(* Logix 5000 project; controller GEA_Test_Chamber vendor 1 type 14 code 196 rev 32.14; software revision 32.04; part 6 of 11 *)
(* tags used below, declared in another part *)
   bPulse05Hz : BOOL;
   bPulse0_1Hz : BOOL;
   bPulse10Hz : BOOL;
   bPulse1Hz : BOOL;
   Cycle_Counter : SINT;
   FVIR_1_S_Step : INT;
   FVIR_1_W_Step : INT;
   FVIR_2_S_Step : INT;
   FVIR_2_W_Step : INT;
   FVIR_3_S_Step : INT;
   FVIR_3_W_Step : INT;
   FVIR_4_S_Step : INT;
   FVIR_4_W_Step : INT;
   FVIR_Gas_Flow_Heater_Indication_1 : BOOL;
   FVIR_Gas_Flow_Heater_Indication_2 : BOOL;
   FVIR_Gas_SCPM_FI001 : REAL;
   FVIR_Gas_SCPM_FI0012 : REAL;
   FVIR_LabView_Comm_OK : BOOL;
   FVIR_Water_Outler_Flow : REAL;
   Gasoline_Step : SINT;
   Mannequin_GoTo_Home : BOOL;
   Mannequin_GoTo_Work : BOOL;
   Mannequin_Step : DINT;
   Pulse : BOOL[32];
   Spill_GoTo_Home : BOOL;
   Spill_GoTo_Work : BOOL;
   Start_Manequinn_Move : BOOL;
   Start_Manequinn_Seq : BOOL;
   Start_Manequinn_Seq_Man : BOOL;
   Start_Spill_Gasoline : BOOL;
   Tigger_First_Manniquine_Seq : BOOL;
   Timer_Delay : TIMER[30];
   tof0_1sPulse : TIMER;
   tof10sPulse : TIMER;
   tof1sPulse : TIMER;
   tof2sPulse : TIMER;
   ton0_1sPulse : TIMER;
   ton10sPulse : TIMER;
   ton1sPulse : TIMER;
   ton2sPulse : TIMER;
   TON_LifeBit_OFF : TIMER;
   TON_LifeBit_ON : TIMER;
   Water_Outlet_Flow_OK : BOOL;
   Water_Outlet_Valve : INT;
   Control_Off : BOOL;
   FVIR_Error_MSG : INT;
   FVIR_LabView_Control : INT;
   FVIR_LabView_Status : INT;
   FVIR_Mannequin_Direction_TimeDelay : INT;
   FVIR_Mannequin_Time_Pause : INT;
   FVIR_Number_Mannequin_Movement : INT;
   FVIR_Reset_Cnt_inprogress : BOOL;
   Output_FVIR : Output_FVIR;
   SET_0 : BOOL;
   SET_1 : BOOL;
(* FVIR_Chamber, continued *)

ROUTINE FVIR_Main   (* ladder *)
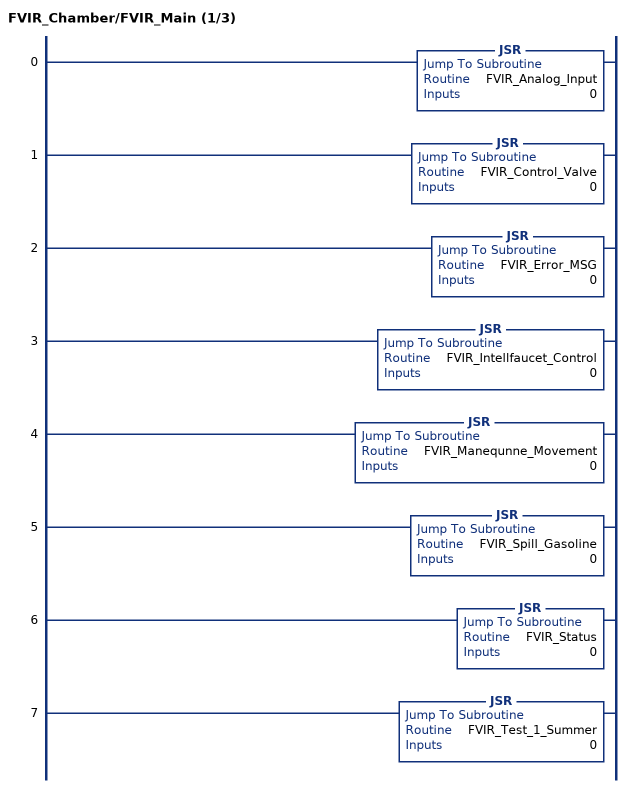
   0: JSR(FVIR_Analog_Input,0);
   1: JSR(FVIR_Control_Valve,0);
   2: JSR(FVIR_Error_MSG,0);
   3: JSR(FVIR_Intellfaucet_Control,0);
   4: JSR(FVIR_Manequnne_Movement,0);
   5: JSR(FVIR_Spill_Gasoline,0);
   6: JSR(FVIR_Status,0);
   7: JSR(FVIR_Test_1_Summer,0);
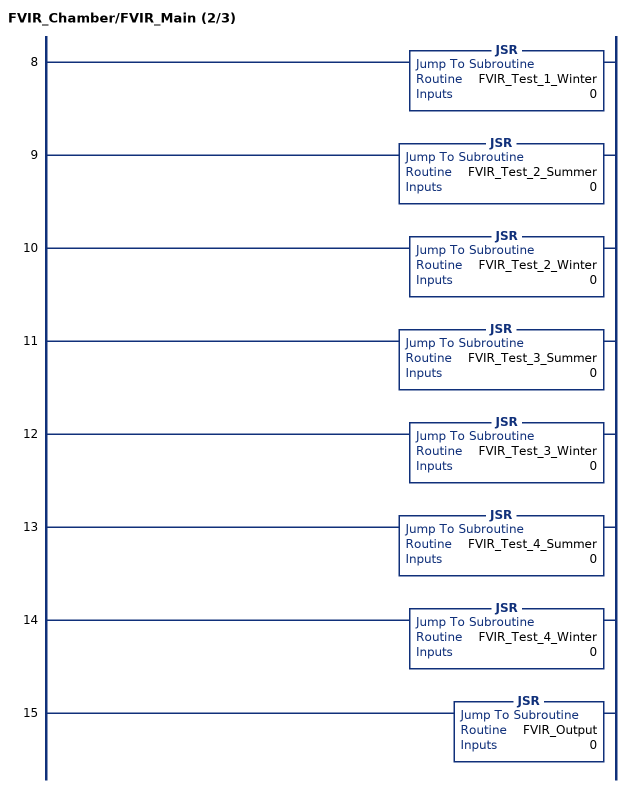
   8: JSR(FVIR_Test_1_Winter,0);
   9: JSR(FVIR_Test_2_Summer,0);
   10: JSR(FVIR_Test_2_Winter,0);
   11: JSR(FVIR_Test_3_Summer,0);
   12: JSR(FVIR_Test_3_Winter,0);
   13: JSR(FVIR_Test_4_Summer,0);
   14: JSR(FVIR_Test_4_Winter,0);
   15: JSR(FVIR_Output,0);
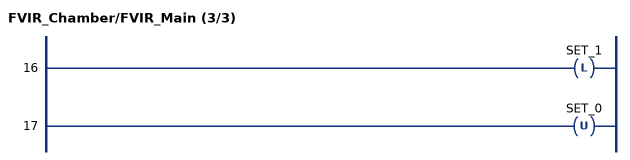
   16: OTL(SET_1);
   17: OTU(SET_0);
END_ROUTINE

ROUTINE FVIR_Manequnne_Movement   (* ladder *)
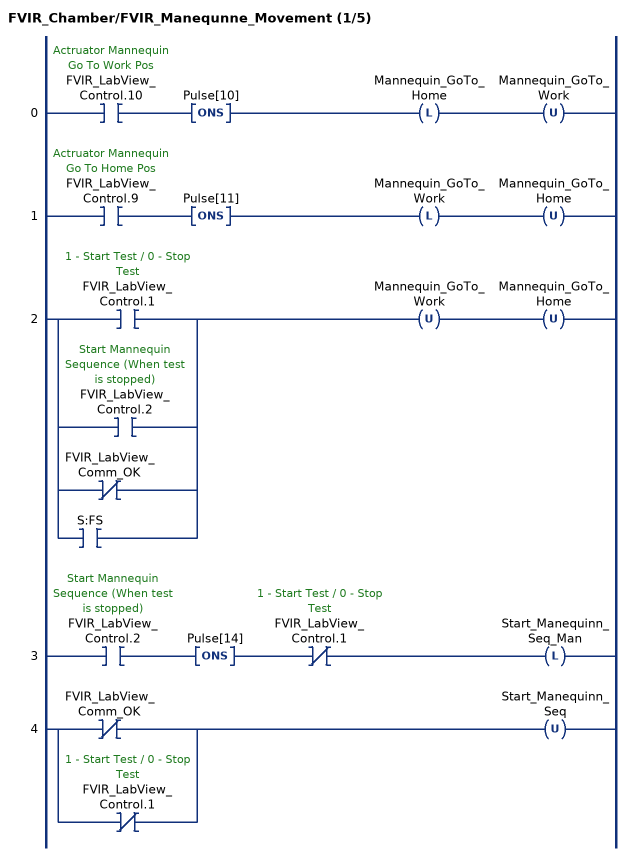
   0: XIC(FVIR_LabView_Control.10)ONS(Pulse[10])OTL(Mannequin_GoTo_Home)OTU(Mannequin_GoTo_Work);
   1: XIC(FVIR_LabView_Control.9)ONS(Pulse[11])OTL(Mannequin_GoTo_Work)OTU(Mannequin_GoTo_Home);
   2: [XIC(FVIR_LabView_Control.1) ,XIC(FVIR_LabView_Control.2) ,[XIO(FVIR_LabView_Comm_OK) ,XIC(S:FS) ] ]OTU(Mannequin_GoTo_Work)OTU(Mannequin_GoTo_Home);
   3: XIC(FVIR_LabView_Control.2)ONS(Pulse[14])XIO(FVIR_LabView_Control.1)OTL(Start_Manequinn_Seq_Man);
   4: [XIO(FVIR_LabView_Comm_OK) ,XIO(FVIR_LabView_Control.1) ]OTU(Start_Manequinn_Seq);
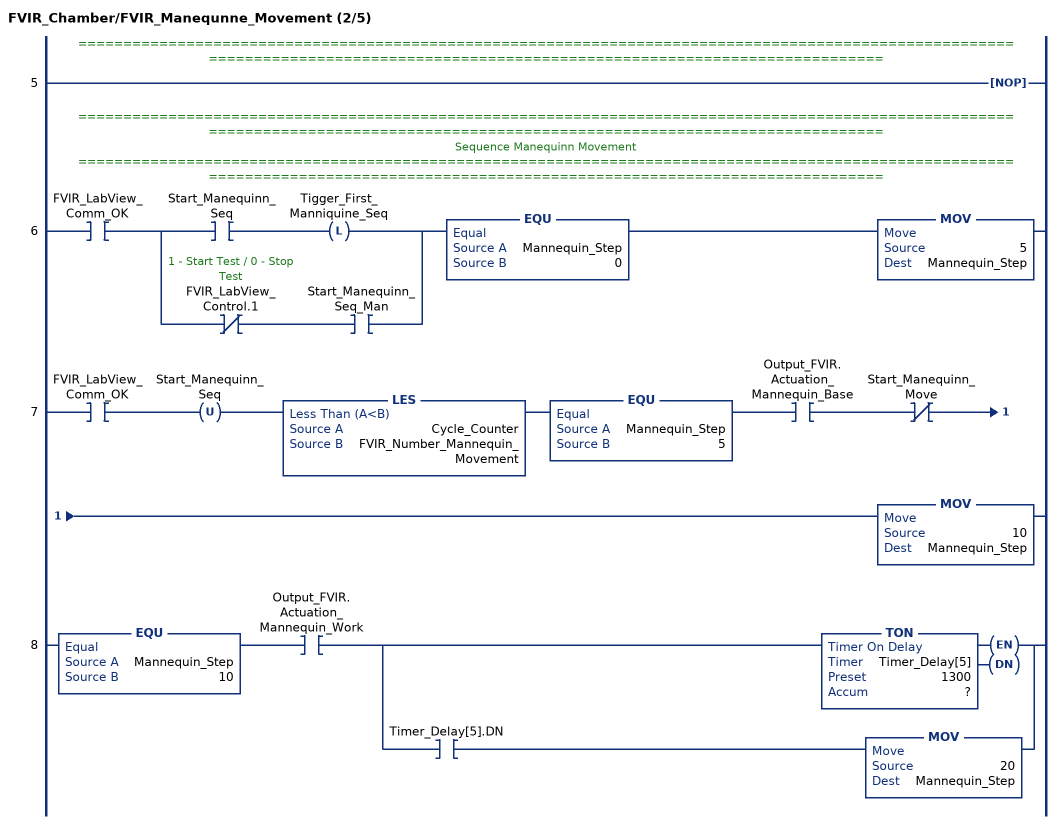
   // ===================================================================================================================================================================================
   5: NOP();
   // ===================================================================================================================================================================================
   // Sequence Manequinn Movement
   // ===================================================================================================================================================================================
   6: XIC(FVIR_LabView_Comm_OK)[XIC(Start_Manequinn_Seq) OTL(Tigger_First_Manniquine_Seq) ,XIO(FVIR_LabView_Control.1) XIC(Start_Manequinn_Seq_Man) ]EQU(Mannequin_Step,0)MOV(5,Mannequin_Step);
   7: XIC(FVIR_LabView_Comm_OK)OTU(Start_Manequinn_Seq)LES(Cycle_Counter,FVIR_Number_Mannequin_Movement)EQU(Mannequin_Step,5)XIC(Output_FVIR.Actuation_Mannequin_Base)XIO(Start_Manequinn_Move)MOV(10,Mannequin_Step);
   8: EQU(Mannequin_Step,10)XIC(Output_FVIR.Actuation_Mannequin_Work)[TON(Timer_Delay[5],?,?) ,XIC(Timer_Delay[5].DN) MOV(20,Mannequin_Step) ];
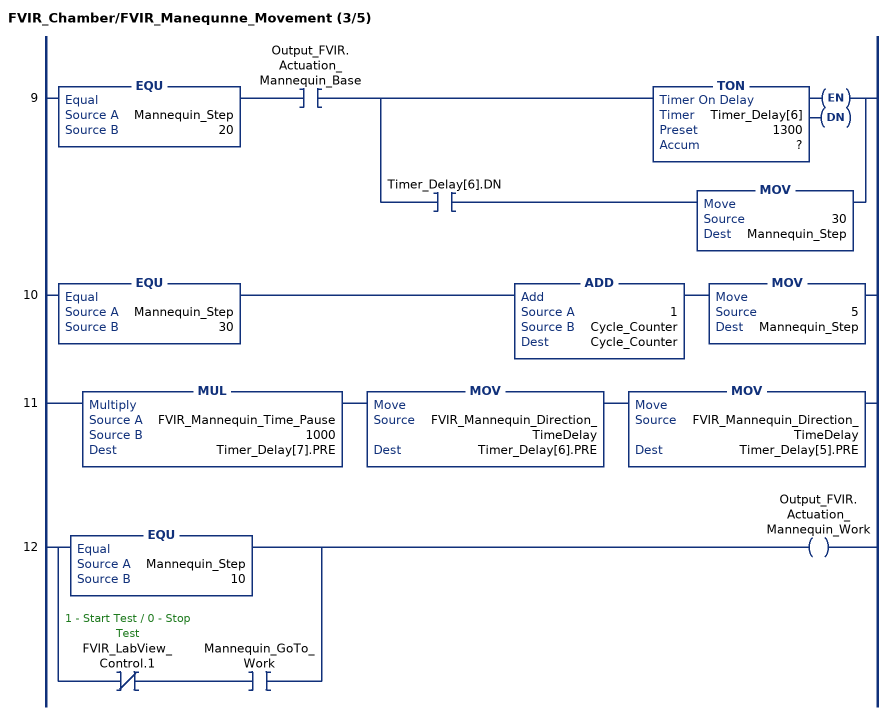
   9: EQU(Mannequin_Step,20)XIC(Output_FVIR.Actuation_Mannequin_Base)[TON(Timer_Delay[6],?,?) ,XIC(Timer_Delay[6].DN) MOV(30,Mannequin_Step) ];
   10: EQU(Mannequin_Step,30)ADD(1,Cycle_Counter,Cycle_Counter)MOV(5,Mannequin_Step);
   11: MUL(FVIR_Mannequin_Time_Pause,1000,Timer_Delay[7].PRE)MOV(FVIR_Mannequin_Direction_TimeDelay,Timer_Delay[6].PRE)MOV(FVIR_Mannequin_Direction_TimeDelay,Timer_Delay[5].PRE);
   12: [EQU(Mannequin_Step,10) ,XIO(FVIR_LabView_Control.1) XIC(Mannequin_GoTo_Work) ]OTE(Output_FVIR.Actuation_Mannequin_Work);
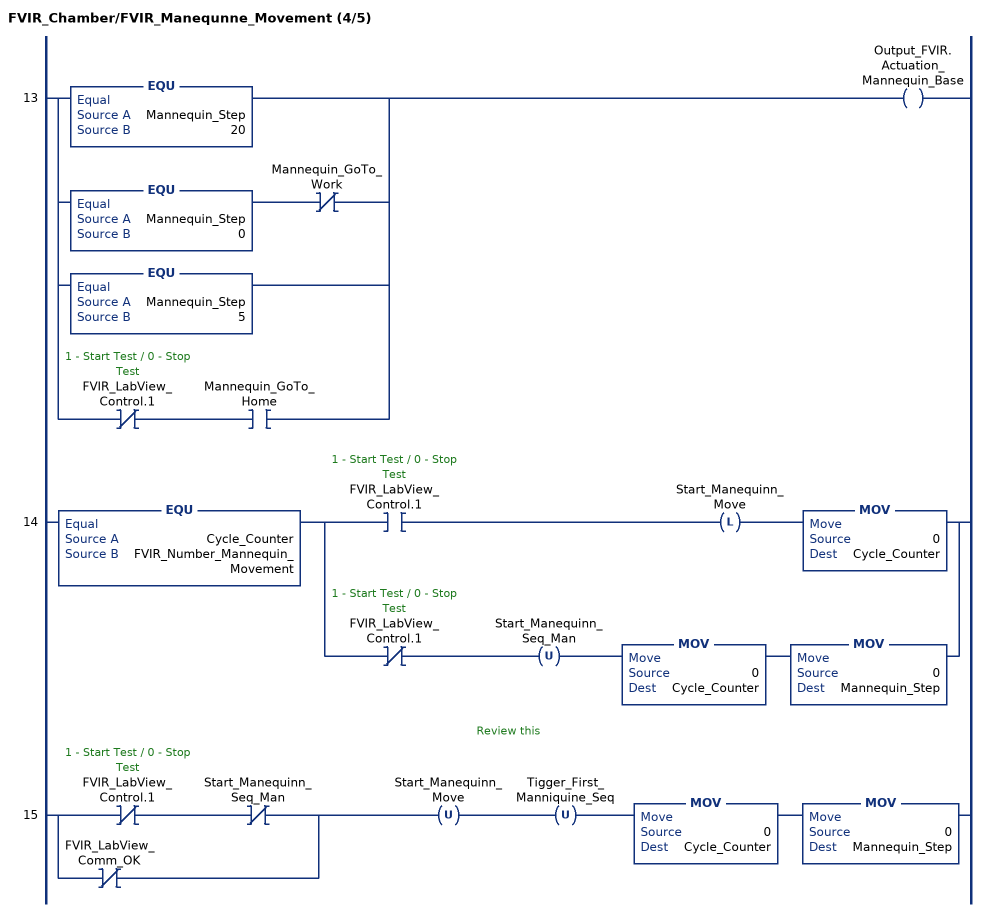
   13: [EQU(Mannequin_Step,20) ,[[EQU(Mannequin_Step,0) XIO(Mannequin_GoTo_Work) ,EQU(Mannequin_Step,5) ] ,XIO(FVIR_LabView_Control.1) XIC(Mannequin_GoTo_Home) ] ]OTE(Output_FVIR.Actuation_Mannequin_Base);
   14: EQU(Cycle_Counter,FVIR_Number_Mannequin_Movement)[XIC(FVIR_LabView_Control.1) OTL(Start_Manequinn_Move) MOV(0,Cycle_Counter) ,XIO(FVIR_LabView_Control.1) OTU(Start_Manequinn_Seq_Man) MOV(0,Cycle_Counter) MOV(0,Mannequin_Step) ];
   // Review this
   15: [XIO(FVIR_LabView_Control.1) XIO(Start_Manequinn_Seq_Man) ,XIO(FVIR_LabView_Comm_OK) ]OTU(Start_Manequinn_Move)OTU(Tigger_First_Manniquine_Seq)MOV(0,Cycle_Counter)MOV(0,Mannequin_Step);
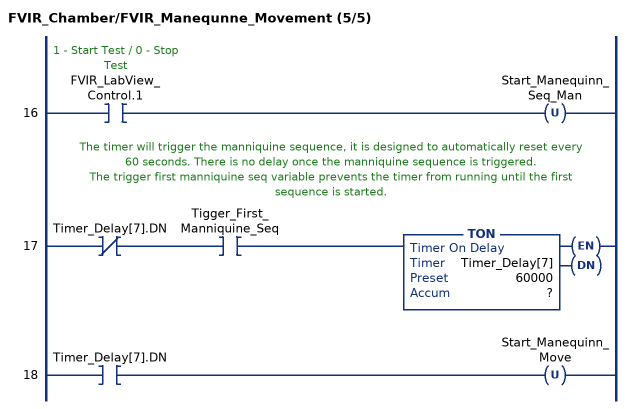
   16: XIC(FVIR_LabView_Control.1)OTU(Start_Manequinn_Seq_Man);
   // The timer will trigger the manniquine sequence, it is designed to automatically reset every 60 seconds. There is no delay once the manniquine sequence is triggered.
   //  The trigger first manniquine seq variable prevents the timer from running until the first sequence is started.
   17: XIO(Timer_Delay[7].DN)XIC(Tigger_First_Manniquine_Seq)TON(Timer_Delay[7],?,?);
   18: XIC(Timer_Delay[7].DN)OTU(Start_Manequinn_Move);
END_ROUTINE

ROUTINE FVIR_Output   (* ladder *)
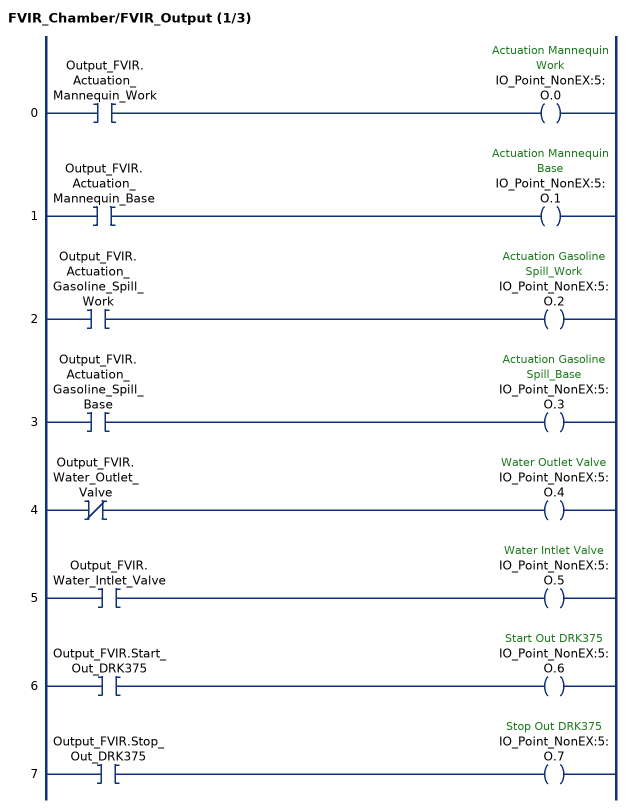
   0: XIC(Output_FVIR.Actuation_Mannequin_Work)OTE(IO_Point_NonEX:5:O.0);
   1: XIC(Output_FVIR.Actuation_Mannequin_Base)OTE(IO_Point_NonEX:5:O.1);
   2: XIC(Output_FVIR.Actuation_Gasoline_Spill_Work)OTE(IO_Point_NonEX:5:O.2);
   3: XIC(Output_FVIR.Actuation_Gasoline_Spill_Base)OTE(IO_Point_NonEX:5:O.3);
   4: XIO(Output_FVIR.Water_Outlet_Valve)OTE(IO_Point_NonEX:5:O.4);
   5: XIC(Output_FVIR.Water_Intlet_Valve)OTE(IO_Point_NonEX:5:O.5);
   6: XIC(Output_FVIR.Start_Out_DRK375)OTE(IO_Point_NonEX:5:O.6);
   7: XIC(Output_FVIR.Stop_Out_DRK375)OTE(IO_Point_NonEX:5:O.7);
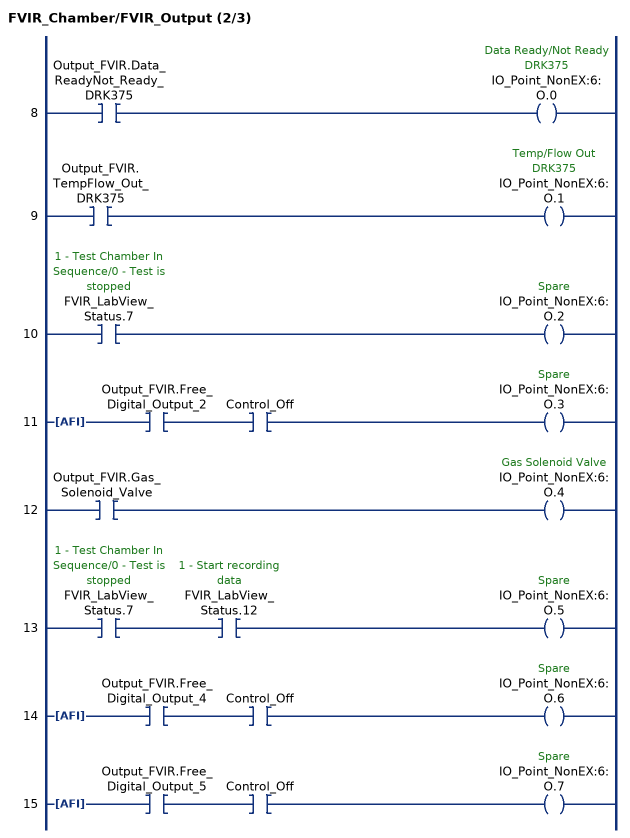
   8: XIC(Output_FVIR.Data_ReadyNot_Ready_DRK375)OTE(IO_Point_NonEX:6:O.0);
   9: XIC(Output_FVIR.TempFlow_Out_DRK375)OTE(IO_Point_NonEX:6:O.1);
   10: XIC(FVIR_LabView_Status.7)OTE(IO_Point_NonEX:6:O.2);
   11: AFI()XIC(Output_FVIR.Free_Digital_Output_2)XIC(Control_Off)OTE(IO_Point_NonEX:6:O.3);
   12: XIC(Output_FVIR.Gas_Solenoid_Valve)OTE(IO_Point_NonEX:6:O.4);
   13: XIC(FVIR_LabView_Status.7)XIC(FVIR_LabView_Status.12)OTE(IO_Point_NonEX:6:O.5);
   14: AFI()XIC(Output_FVIR.Free_Digital_Output_4)XIC(Control_Off)OTE(IO_Point_NonEX:6:O.6);
   15: AFI()XIC(Output_FVIR.Free_Digital_Output_5)XIC(Control_Off)OTE(IO_Point_NonEX:6:O.7);
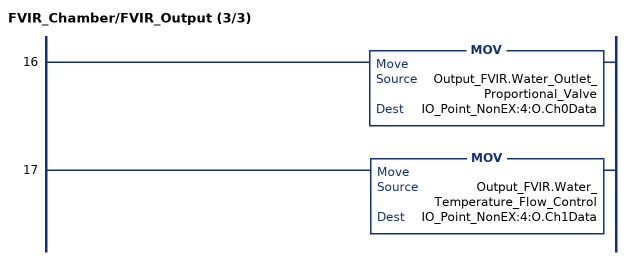
   16: MOV(Output_FVIR.Water_Outlet_Proportional_Valve,IO_Point_NonEX:4:O.Ch0Data);
   17: MOV(Output_FVIR.Water_Temperature_Flow_Control,IO_Point_NonEX:4:O.Ch1Data);
END_ROUTINE

ROUTINE FVIR_Spill_Gasoline   (* ladder *)
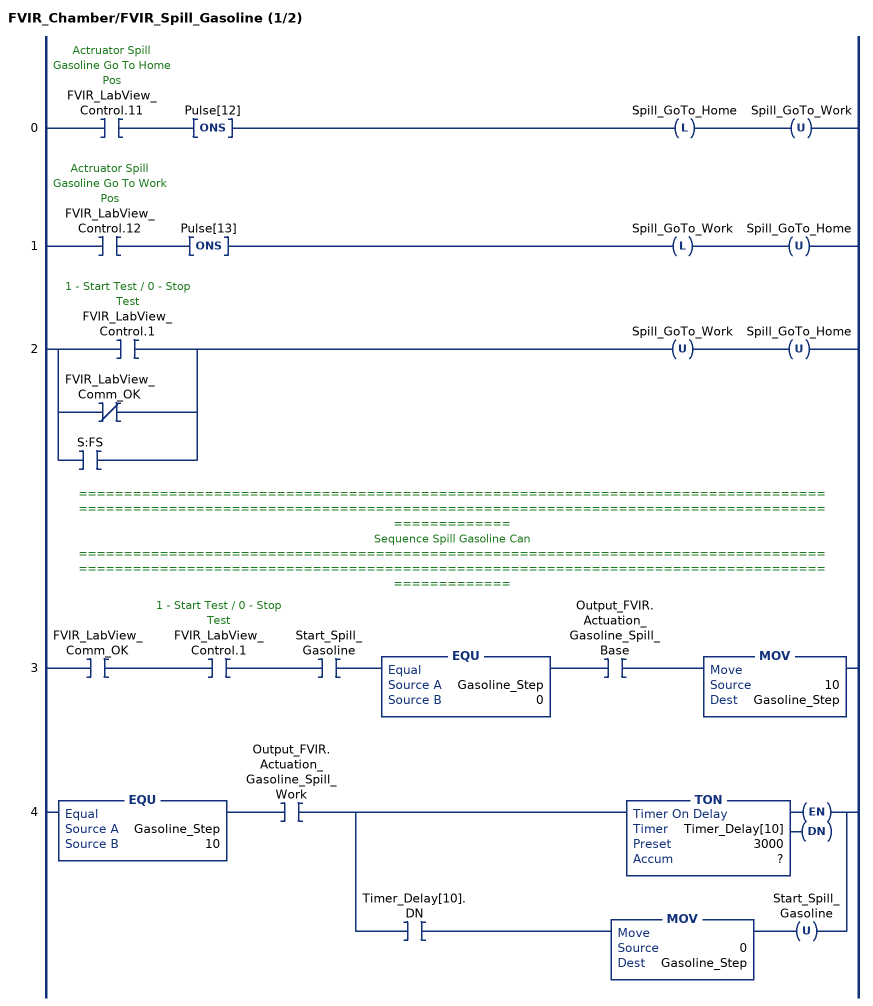
   0: XIC(FVIR_LabView_Control.11)ONS(Pulse[12])OTL(Spill_GoTo_Home)OTU(Spill_GoTo_Work);
   1: XIC(FVIR_LabView_Control.12)ONS(Pulse[13])OTL(Spill_GoTo_Work)OTU(Spill_GoTo_Home);
   2: [XIC(FVIR_LabView_Control.1) ,[XIO(FVIR_LabView_Comm_OK) ,XIC(S:FS) ] ]OTU(Spill_GoTo_Work)OTU(Spill_GoTo_Home);
   // ===================================================================================================================================================================================
   // Sequence Spill Gasoline Can
   // ===================================================================================================================================================================================
   3: XIC(FVIR_LabView_Comm_OK)XIC(FVIR_LabView_Control.1)XIC(Start_Spill_Gasoline)EQU(Gasoline_Step,0)XIC(Output_FVIR.Actuation_Gasoline_Spill_Base)MOV(10,Gasoline_Step);
   4: EQU(Gasoline_Step,10)XIC(Output_FVIR.Actuation_Gasoline_Spill_Work)[TON(Timer_Delay[10],?,?) ,XIC(Timer_Delay[10].DN) MOV(0,Gasoline_Step) OTU(Start_Spill_Gasoline) ];
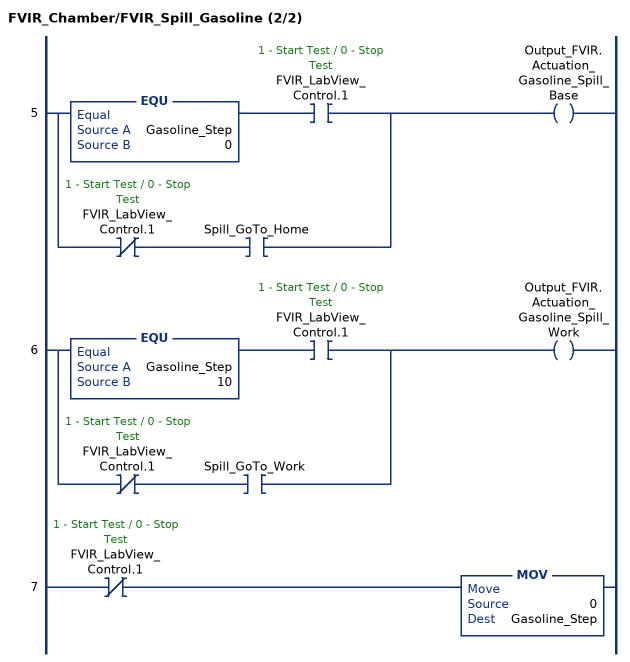
   5: [EQU(Gasoline_Step,0) XIC(FVIR_LabView_Control.1) ,XIO(FVIR_LabView_Control.1) XIC(Spill_GoTo_Home) ]OTE(Output_FVIR.Actuation_Gasoline_Spill_Base);
   6: [EQU(Gasoline_Step,10) XIC(FVIR_LabView_Control.1) ,XIO(FVIR_LabView_Control.1) XIC(Spill_GoTo_Work) ]OTE(Output_FVIR.Actuation_Gasoline_Spill_Work);
   7: XIO(FVIR_LabView_Control.1)MOV(0,Gasoline_Step);
END_ROUTINE

ROUTINE FVIR_Status   (* ladder *)
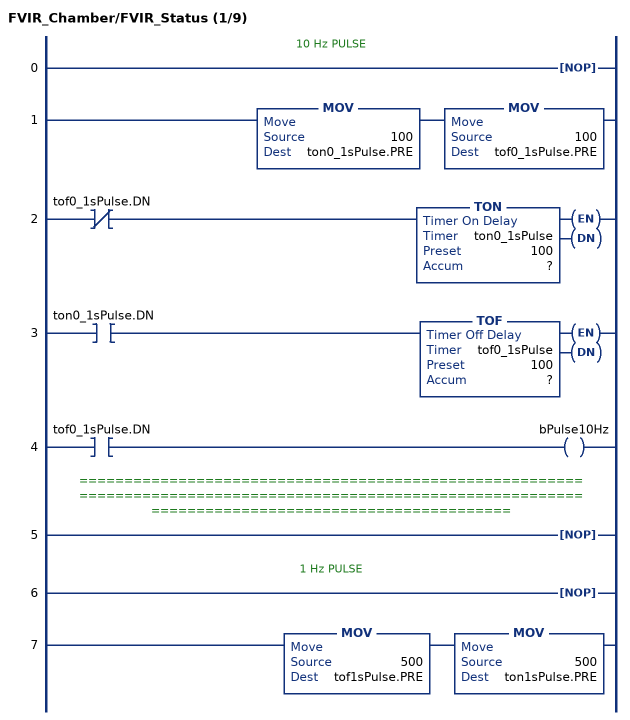
   // 10 Hz PULSE
   0: NOP();
   1: MOV(100,ton0_1sPulse.PRE)MOV(100,tof0_1sPulse.PRE);
   2: XIO(tof0_1sPulse.DN)TON(ton0_1sPulse,?,?);
   3: XIC(ton0_1sPulse.DN)TOF(tof0_1sPulse,?,?);
   4: XIC(tof0_1sPulse.DN)OTE(bPulse10Hz);
   // ========================================================================================================================================================
   5: NOP();
   // 1 Hz PULSE
   6: NOP();
   7: MOV(500,tof1sPulse.PRE)MOV(500,ton1sPulse.PRE);
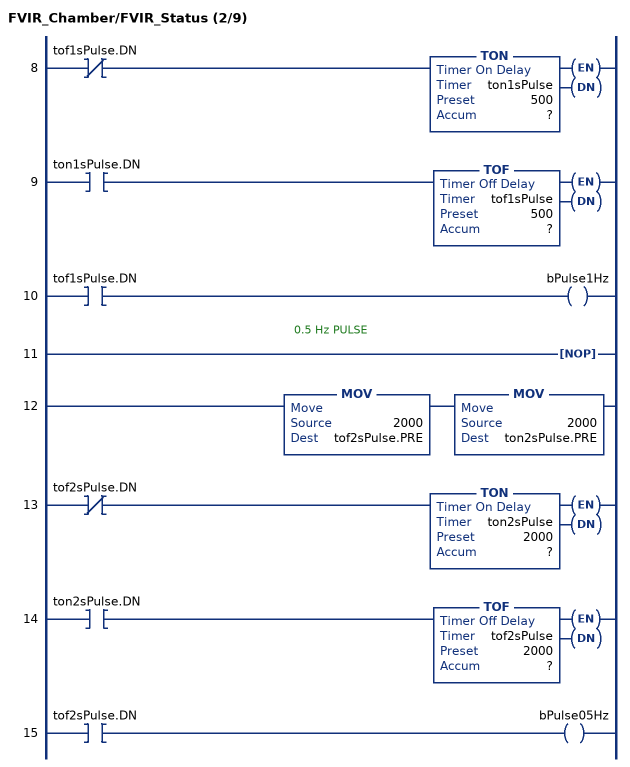
   8: XIO(tof1sPulse.DN)TON(ton1sPulse,?,?);
   9: XIC(ton1sPulse.DN)TOF(tof1sPulse,?,?);
   10: XIC(tof1sPulse.DN)OTE(bPulse1Hz);
   // 0.5 Hz PULSE
   11: NOP();
   12: MOV(2000,tof2sPulse.PRE)MOV(2000,ton2sPulse.PRE);
   13: XIO(tof2sPulse.DN)TON(ton2sPulse,?,?);
   14: XIC(ton2sPulse.DN)TOF(tof2sPulse,?,?);
   15: XIC(tof2sPulse.DN)OTE(bPulse05Hz);
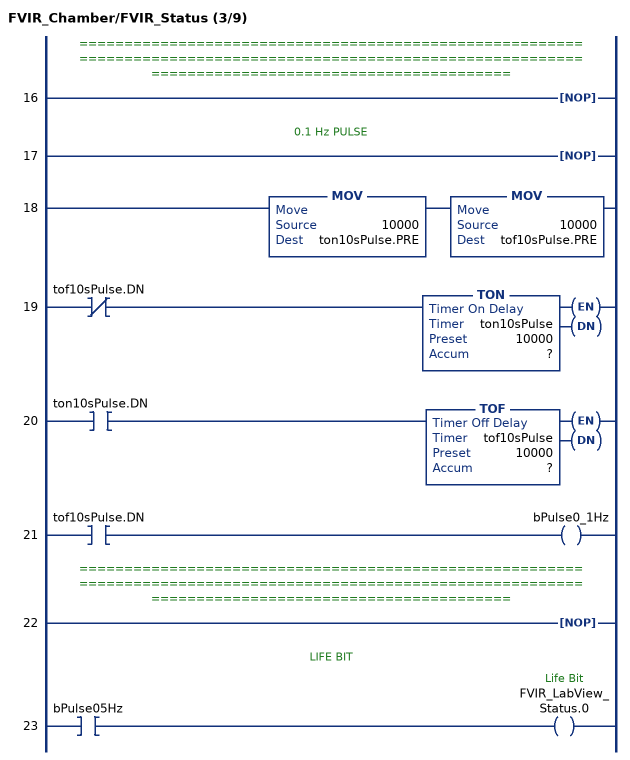
   // ========================================================================================================================================================
   16: NOP();
   // 0.1 Hz PULSE
   17: NOP();
   18: MOV(10000,ton10sPulse.PRE)MOV(10000,tof10sPulse.PRE);
   19: XIO(tof10sPulse.DN)TON(ton10sPulse,?,?);
   20: XIC(ton10sPulse.DN)TOF(tof10sPulse,?,?);
   21: XIC(tof10sPulse.DN)OTE(bPulse0_1Hz);
   // ========================================================================================================================================================
   22: NOP();
   // LIFE BIT
   23: XIC(bPulse05Hz)OTE(FVIR_LabView_Status.0);
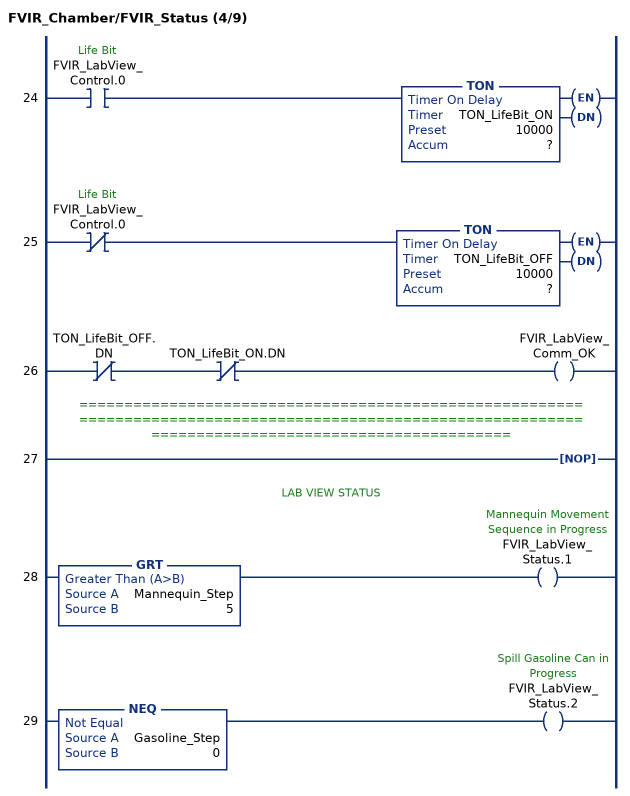
   24: XIC(FVIR_LabView_Control.0)TON(TON_LifeBit_ON,?,?);
   25: XIO(FVIR_LabView_Control.0)TON(TON_LifeBit_OFF,?,?);
   26: XIO(TON_LifeBit_OFF.DN)XIO(TON_LifeBit_ON.DN)OTE(FVIR_LabView_Comm_OK);
   // ========================================================================================================================================================
   27: NOP();
   // LAB VIEW STATUS
   28: GRT(Mannequin_Step,5)OTE(FVIR_LabView_Status.1);
   29: NEQ(Gasoline_Step,0)OTE(FVIR_LabView_Status.2);
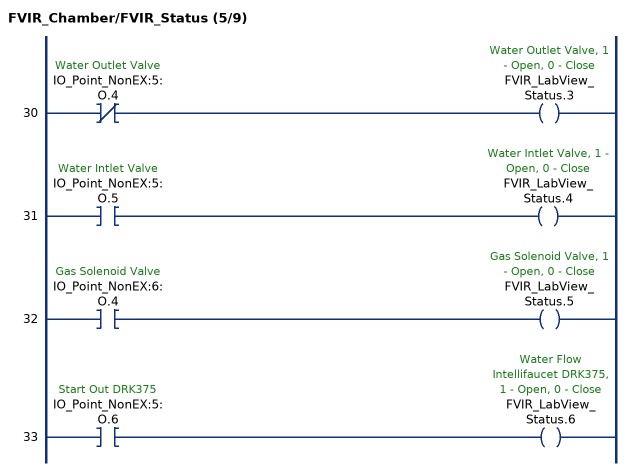
   30: XIO(IO_Point_NonEX:5:O.4)OTE(FVIR_LabView_Status.3);
   31: XIC(IO_Point_NonEX:5:O.5)OTE(FVIR_LabView_Status.4);
   32: XIC(IO_Point_NonEX:6:O.4)OTE(FVIR_LabView_Status.5);
   33: XIC(IO_Point_NonEX:5:O.6)OTE(FVIR_LabView_Status.6);
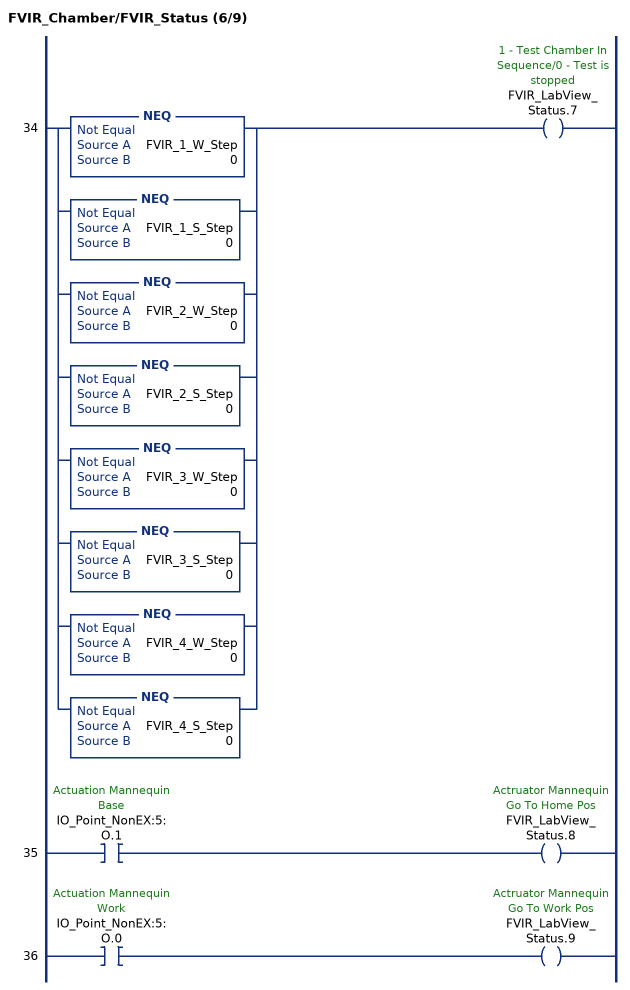
   34: [NEQ(FVIR_1_W_Step,0) ,NEQ(FVIR_1_S_Step,0) ,NEQ(FVIR_2_W_Step,0) ,NEQ(FVIR_2_S_Step,0) ,NEQ(FVIR_3_W_Step,0) ,NEQ(FVIR_3_S_Step,0) ,NEQ(FVIR_4_W_Step,0) ,NEQ(FVIR_4_S_Step,0) ]OTE(FVIR_LabView_Status.7);
   35: XIC(IO_Point_NonEX:5:O.1)OTE(FVIR_LabView_Status.8);
   36: XIC(IO_Point_NonEX:5:O.0)OTE(FVIR_LabView_Status.9);
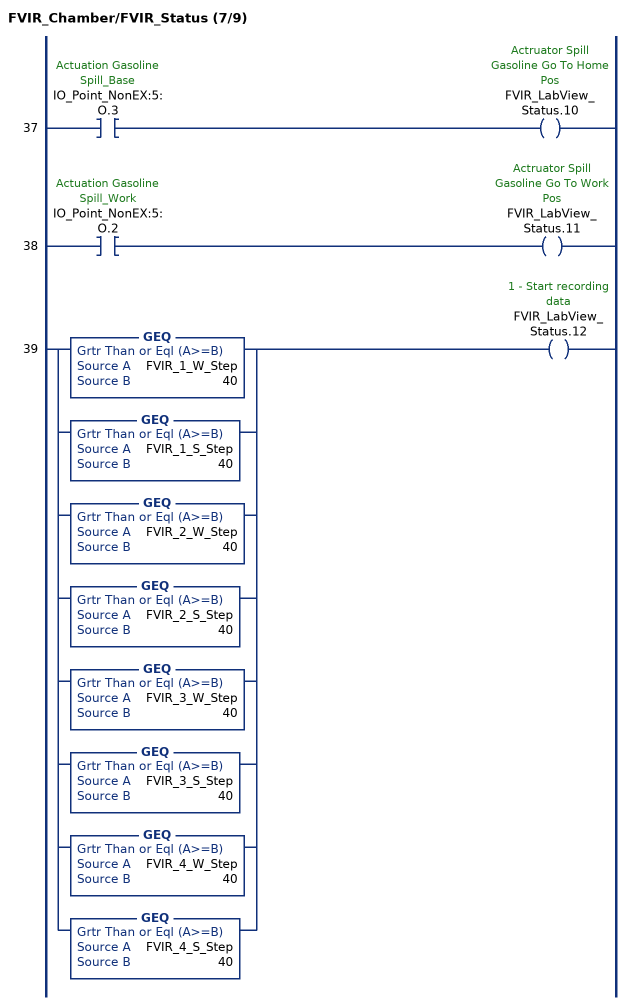
   37: XIC(IO_Point_NonEX:5:O.3)OTE(FVIR_LabView_Status.10);
   38: XIC(IO_Point_NonEX:5:O.2)OTE(FVIR_LabView_Status.11);
   39: [GEQ(FVIR_1_W_Step,40) ,GEQ(FVIR_1_S_Step,40) ,GEQ(FVIR_2_W_Step,40) ,GEQ(FVIR_2_S_Step,40) ,GEQ(FVIR_3_W_Step,40) ,GEQ(FVIR_3_S_Step,40) ,GEQ(FVIR_4_W_Step,40) ,GEQ(FVIR_4_S_Step,40) ]OTE(FVIR_LabView_Status.12);
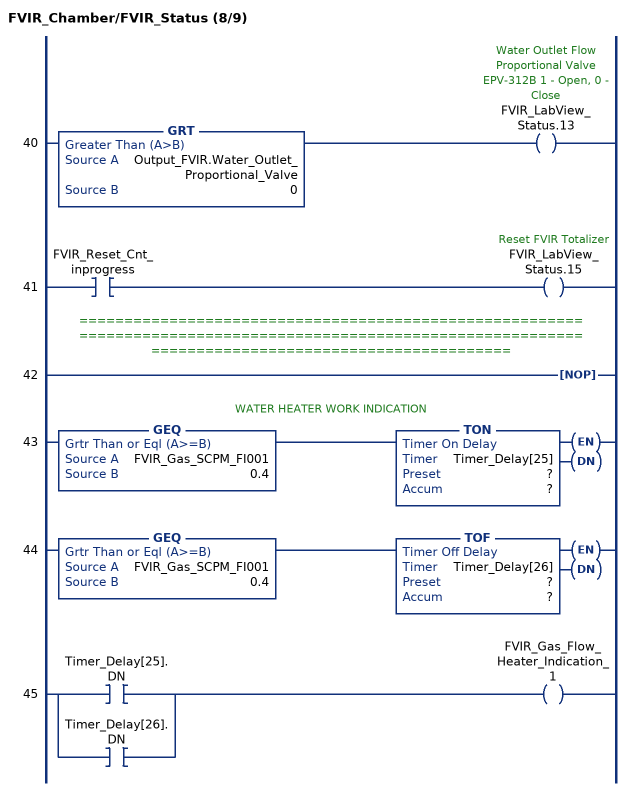
   40: GRT(Output_FVIR.Water_Outlet_Proportional_Valve,0)OTE(FVIR_LabView_Status.13);
   41: XIC(FVIR_Reset_Cnt_inprogress)OTE(FVIR_LabView_Status.15);
   // ========================================================================================================================================================
   42: NOP();
   // WATER HEATER WORK INDICATION
   43: GEQ(FVIR_Gas_SCPM_FI001,0.4)TON(Timer_Delay[25],?,?);
   44: GEQ(FVIR_Gas_SCPM_FI001,0.4)TOF(Timer_Delay[26],?,?);
   45: [XIC(Timer_Delay[25].DN) ,XIC(Timer_Delay[26].DN) ]OTE(FVIR_Gas_Flow_Heater_Indication_1);
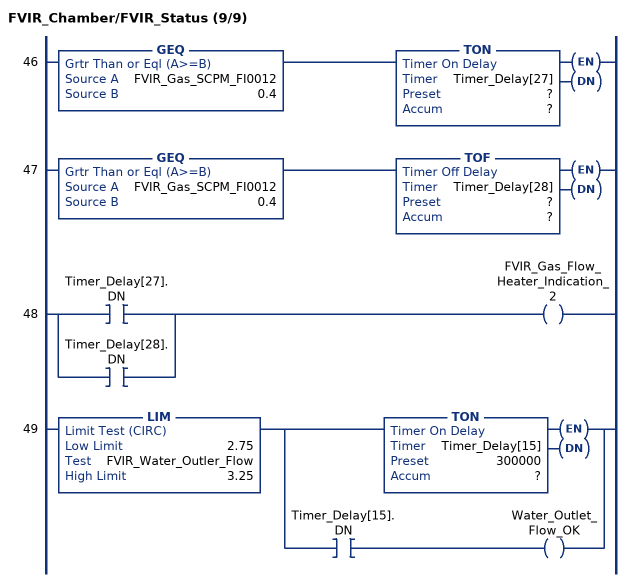
   46: GEQ(FVIR_Gas_SCPM_FI0012,0.4)TON(Timer_Delay[27],?,?);
   47: GEQ(FVIR_Gas_SCPM_FI0012,0.4)TOF(Timer_Delay[28],?,?);
   48: [XIC(Timer_Delay[27].DN) ,XIC(Timer_Delay[28].DN) ]OTE(FVIR_Gas_Flow_Heater_Indication_2);
   49: LIM(2.75,FVIR_Water_Outler_Flow,3.25)[TON(Timer_Delay[15],?,?) ,XIC(Timer_Delay[15].DN) OTE(Water_Outlet_Flow_OK) ];
END_ROUTINE
